FUNCTION_BLOCK MultipleChangeDetect (* Composite Function Block Type *)
  (* Standard: 61499-2 *)
  (* Version 0.0, 11/1/2016, chivdan, nxtControl GmbH, template *)
  PACKAGE Main;
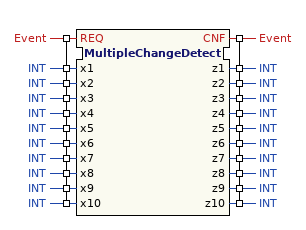
  EVENT_INPUT
    REQ WITH x1, x2, x3, x4, x5, x7, x6, x8, x9, x10; (* Normal Execution Request *)
  END_EVENT
  EVENT_OUTPUT
    CNF WITH z1, z2, z3, z4, z5, z6, z7, z8, z9, z10; (* Execution Confirmation *)
  END_EVENT
  VAR_INPUT
    x1 : INT; (* Input event qualifier *)
    x2 : INT;
    x3 : INT;
    x4 : INT;
    x5 : INT;
    x6 : INT;
    x7 : INT;
    x8 : INT;
    x9 : INT;
    x10 : INT;
  END_VAR
  VAR_OUTPUT
    z1 : INT; (* Output event qualifier *)
    z2 : INT;
    z3 : INT;
    z4 : INT;
    z5 : INT;
    z6 : INT;
    z7 : INT;
    z8 : INT;
    z9 : INT;
    z10 : INT;
  END_VAR
  FBS
    FB1 : E_D_FF;
    FB2 : E_D_FF;
    FB3 : E_D_FF;
    FB4 : E_D_FF;
    FB5 : E_D_FF;
    FB6 : E_D_FF;
    FB7 : E_D_FF;
    FB8 : E_D_FF;
    FB9 : E_D_FF;
    FB10 : E_D_FF;
    FB11 : MultipleEMerge;
  END_FBS
  EVENT_CONNECTIONS
    REQ TO FB1.CLK;
    REQ TO FB2.CLK;
    REQ TO FB3.CLK;
    REQ TO FB4.CLK;
    REQ TO FB5.CLK;
    REQ TO FB6.CLK;
    REQ TO FB7.CLK;
    REQ TO FB8.CLK;
    REQ TO FB9.CLK;
    FB1.EO TO FB11.REQ1;
    FB2.EO TO FB11.REQ2;
    FB3.EO TO FB11.REQ3;
    FB4.EO TO FB11.REQ4;
    FB5.EO TO FB11.REQ5;
    FB6.EO TO FB11.REQ6;
    FB7.EO TO FB11.REQ7;
    FB8.EO TO FB11.REQ8;
    FB9.EO TO FB11.REQ9;
    FB10.EO TO FB11.REQ10;
    FB11.CNF TO CNF;
  END_CONNECTIONS
  DATA_CONNECTIONS
    x1 TO FB1.D;
    x2 TO FB2.D;
    x3 TO FB3.D;
    x4 TO FB4.D;
    x5 TO FB5.D;
    x6 TO FB6.D;
    x7 TO FB7.D;
    x8 TO FB8.D;
    x9 TO FB9.D;
    x10 TO FB10.D;
    FB1.Q TO z1;
    FB2.Q TO z2;
    FB3.Q TO z3;
    FB4.Q TO z4;
    FB5.Q TO z5;
    FB6.Q TO z6;
    FB7.Q TO z7;
    FB8.Q TO z8;
    FB9.Q TO z9;
    FB10.Q TO z10;
  END_CONNECTIONS
END_FUNCTION_BLOCK
